(* IEC 61131-3 sources: cs6494-fall2026-students/labs/substation-recovery-demo/st, 4 files *)

(* ---- deny_all.st ---- *)
FUNCTION CloseInterlock : BOOL
VAR_INPUT
  CloseRequested : BOOL;
  ActualPositions : BYTE;
  TargetMask : BYTE;
  OutOfServiceMask : BYTE;
  TripLatched : BOOL;
  PresentCurrent_dA : UINT;
  CurrentLimit_dA : UINT;
END_VAR

(* Faulty patch: safe from closing, but incapable of restoring service. *)
CloseInterlock := FALSE;
END_FUNCTION

(* ---- repaired.st ---- *)
FUNCTION CloseInterlock : BOOL
VAR_INPUT
  CloseRequested : BOOL;
  ActualPositions : BYTE;
  TargetMask : BYTE;
  OutOfServiceMask : BYTE;
  TripLatched : BOOL;
  PresentCurrent_dA : UINT;
  CurrentLimit_dA : UINT;
END_VAR
VAR
  ProjectedPositions : BYTE;
  EnergizedBranches : BYTE;
END_VAR

(* Repair: decide from the topology that would result after the request. *)
ProjectedPositions := ActualPositions OR TargetMask;

IF (ProjectedPositions AND 16#01) <> 0 THEN
  EnergizedBranches := ProjectedPositions AND 16#0E;
ELSE
  EnergizedBranches := 0;
END_IF;

CloseInterlock :=
  CloseRequested
  AND NOT TripLatched
  AND ((EnergizedBranches AND OutOfServiceMask) = 0);
END_FUNCTION

(* ---- target_local.st ---- *)
FUNCTION CloseInterlock : BOOL
VAR_INPUT
  CloseRequested : BOOL;
  ActualPositions : BYTE;
  TargetMask : BYTE;
  OutOfServiceMask : BYTE;
  TripLatched : BOOL;
  PresentCurrent_dA : UINT;
  CurrentLimit_dA : UINT;
END_VAR

(* Faulty patch: blocks only a command whose named target is out of service. *)
CloseInterlock :=
  CloseRequested
  AND NOT TripLatched
  AND ((TargetMask AND OutOfServiceMask) = 0)
  AND (PresentCurrent_dA < CurrentLimit_dA);
END_FUNCTION

(* ---- vulnerable.st ---- *)
FUNCTION CloseInterlock : BOOL
VAR_INPUT
  CloseRequested : BOOL;
  ActualPositions : BYTE;
  TargetMask : BYTE;
  OutOfServiceMask : BYTE;
  TripLatched : BOOL;
  PresentCurrent_dA : UINT;
  CurrentLimit_dA : UINT;
END_VAR

(* Vulnerable: present current does not predict the proposed topology. *)
CloseInterlock :=
  CloseRequested
  AND NOT TripLatched
  AND (PresentCurrent_dA < CurrentLimit_dA);
END_FUNCTION
